FUNCTION F_LogWarning : T_MaxString 
VAR_INPUT
    Message : T_MaxString;
END_VAR

ADSLOGSTR(
    msgCtrlMask := ADSLOG_MSGTYPE_STRING OR ADSLOG_MSGTYPE_WARN OR ADSLOG_MSGTYPE_LOG,
    msgFmtStr := Message,
    strArg := '');

END_FUNCTION

(* stored: Version 1.1.0.1, ProductVersion 3.1.4024.3
   POU F_LogWarning: Id {e17ba9d2-e637-06e2-2c27-e11fe52482dd}, SpecialFunc None *)
